{attribute 'TcGenerated'}
{attribute 'no-analysis'}
{attribute 'linkalways'}
// This function has been automatically generated from the project information.
VAR_GLOBAL CONSTANT
	{attribute 'const_non_replaced'}
	stLibVersion_tcl_SimpleUnitTestLibrary : ST_LibVersion := (iMajor := 1, iMinor := 1, iBuild := 4, iRevision := 0, nFlags := 0, sVersion := '1.1.4.0');
END_VAR

(* stored: Version 1.1.0.1, ProductVersion 3.1.4024.6
   GVL Global_Version: Id {7a4531ca-e3f3-43ce-ae6c-8653b5fea95b} *)
